RoboDK station: demo.rdk

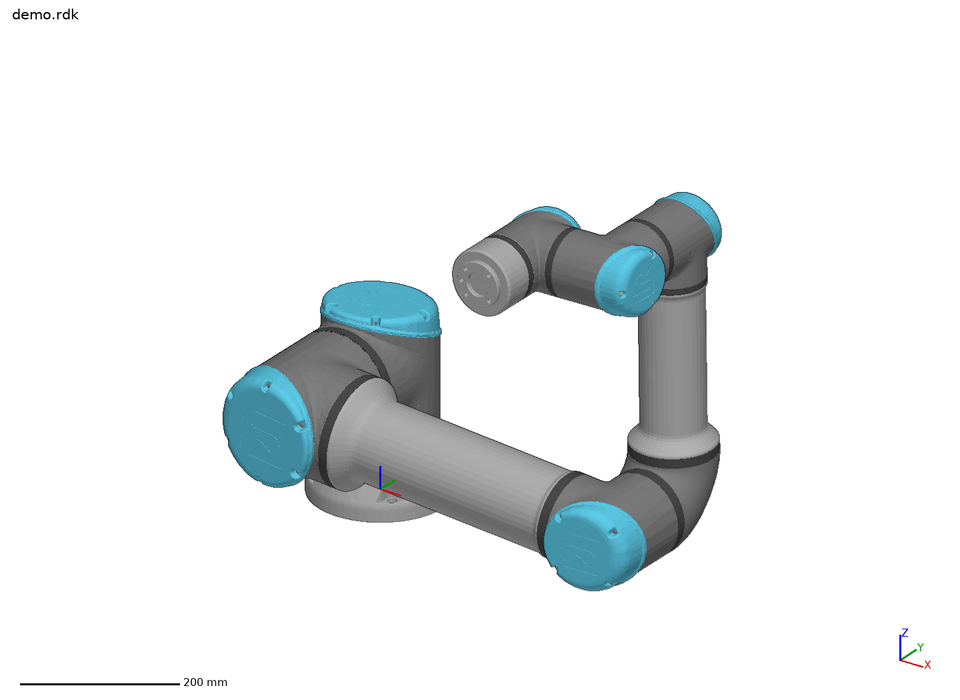
[picture v0: the station drawn from its stored meshes, robots at their saved joint values, targets as dots, program paths as lines]
Station demo (saved by RoboDK 5.7.4). Poses are relative to the parent item; angles as X-Y-Z fixed-axis rotations.
  - frame UR16e Base at (0, 0, 0) mm
    - robot UR16e: 6 axes, payload 16 kg, reach 900 mm, repeatability 0.05 mm, weight 33.1 kg
        modified DH rows (alpha deg, a mm, theta deg, d mm): 0, 0, 0, 180.7; 90, 0, 180, 0; 0, 478.4, 0, 0; 0, 360, 0, 174.15; -90, 0, 0, 119.85; 90, 0, 180, 116.55
        joint limits [-360, -360, -360, -360, -360, -360] to [360, 360, 360, 360, 360, 360]; home [0, -90, -90, 0, 90, 0]; saved at [0, 175.231, -264.431, 0, 0, 0]
  - Python program Prog1 (listed below)

--- Python program Prog1 ---
from robolink import *    # RoboDK API
from robodk import *      # Robot toolbox
import paho.mqtt.client as mqtt
import time
import random
import json
import numpy as np

print("starting...")

RL = Robolink()

robot = RL.Item('UR16e')
#joint_angles = [math.radians(45), math.radians(-30), math.radians(60), math.radians(-45), math.radians(30), math.radians(0)]

# Move the robot to the specified joint angles using joint movement
#robot.MoveJ(joint_angles)

# Define another set of joint angles
#joint_angles_2 = [math.radians(-45), math.radians(30), math.radians(-60), math.radians(45), math.radians(-30), math.radians(90)]

# Move the robot to the new set of joint angles using joint movement
#robot.MoveJ(joint_angles_2)
robot.MoveJ([0, 0, 0, 0, 0, 0])
mediapipe_topic = 'mediapipe'

def cartesian_to_cylindrical_3d(data):
    x, y, z = data[0], data[1], data[2]
    r = math.sqrt(x**2 + y**2)
    theta = math.atan2(y, x)
    return r, theta, z

def on_connect(client, userdata, flags, rc, properties):
    print(f"Connected with result code {rc}-----------------------------")
    client.subscribe('mediapipe')
    #client.subscribe(MQTT_METADATA['motiontopic'])

prev_shoulder = 0
prev_elbow = 0
prev_wrist = 0

def on_message(client, userdata, message):
    data = json.loads(message.payload.decode())
    data = np.asarray(data)
    _, shoulder, z_shoulder = cartesian_to_cylindrical_3d(data[1] - data[0])
    _, elbow, z_elbow = cartesian_to_cylindrical_3d(data[2] - data[1])
    _, wrist, z_wrist = cartesian_to_cylindrical_3d(data[2])

    if data[0][3] < 0.5:
        shoulder = prev_shoulder
    else:
        prev_shoulder = shoulder
    if data[1][3] < 0.5:
        elbow = prev_shoulder
    else:
        prev_elbow = elbow


    elbow = elbow - shoulder
    wrist = wrist - elbow - shoulder
    #print(f"Joints {shoulder}, {elbow}, {wrist}")
    #print(f"Joints {data[0]}, {data[1]}, {math.degrees(elbow)}")
    robot.MoveJ([0, math.degrees(shoulder), math.degrees(elbow), 0, 0, 0])
    #time.sleep(1/100)

print("connecting to mqtt")
client_id = f'python-mqtt-{random.randint(0, 1000)}'
#client = mqtt.Client(mqtt.CallbackAPIVersion.VERSION2, transport='websockets')
client = mqtt.Client(mqtt.CallbackAPIVersion.VERSION2, transport="websockets")

client.on_connect = on_connect
client.on_message = on_message

# was port 9001
client.connect('localhost', 8080, 60)  # 60 is waiting interval
client.loop_forever()

# Define the MQTT topic

"""
# Initialize the RoboDK API
if __name__ == '__main__':

    RL = Robolink()

    robot = RL.Item('UR16e')
    joint_angles = [math.radians(45), math.radians(-30), math.radians(60), math.radians(-45), math.radians(30), math.radians(0)]

    # Move the robot to the specified joint angles using joint movement
    robot.MoveJ(joint_angles)

    # Define another set of joint angles
    joint_angles_2 = [math.radians(-45), math.radians(30), math.radians(-60), math.radians(45), math.radians(-30), math.radians(90)]

    # Move the robot to the new set of joint angles using joint movement
    robot.MoveJ(joint_angles_2)
"""
